(* PLC project Unnamed, Unknown Unnamed 1 *)
(* stored: creationDateTime 2023-06-20T15:59:41, modificationDateTime 2023-06-21T09:28:57 *)

PROGRAM filling_tank
  VAR
    manual AT %QX0.0 : BOOL;
    auto AT %QX0.1 : BOOL;
    emergency_stop AT %QX0.2 : BOOL;
    start AT %QX0.3 : BOOL;
    stop AT %QX0.4 : BOOL;
    reset_button AT %QX0.5 : BOOL;
    start_light AT %QX1.0 : BOOL;
    stop_light AT %QX1.1 : BOOL;
    reset_light AT %QX1.2 : BOOL;
    bottom_valve_open AT %QX1.3 : BOOL;
    top_valve_open AT %QX1.4 : BOOL;
    fictoryioreset AT %QX1.5 : BOOL;
    top_flow AT %QW0 : INT;
    top_level AT %QW1 : INT;
    bottom_flow AT %QW2 : INT;
    bottom_level AT %QW3 : INT;
    top_fill_valve AT %QW4 : INT;
    top_discharge_valve AT %QW5 : INT;
    bottom_fill_valve AT %QW6 : INT;
    bottom_discharge_valve AT %QW7 : INT;
    top_tank AT %QW8 : INT;
    bottom_tank AT %QW9 : INT;
    number_cycles AT %QW10 : INT;
  END_VAR
  VAR
    CTU0 : CTU;
    reset : BOOL;
  END_VAR
  VAR  (* added by the conversion: wires and edge detectors of the diagram *)
    _MOVE9_ENO : BOOL;
    _MOVE9_OUT : INT;
    _LT31_ENO : BOOL;
    _LT31_OUT : BOOL;
    _LT32_ENO : BOOL;
    _LT32_OUT : BOOL;
    _MOVE36_ENO : BOOL;
    _MOVE36_OUT : INT;
    _MOVE38_ENO : BOOL;
    _MOVE38_OUT : INT;
    _GT19_ENO : BOOL;
    _GT19_OUT : BOOL;
    _MOVE22_ENO : BOOL;
    _MOVE22_OUT : INT;
    _MOVE24_ENO : BOOL;
    _MOVE24_OUT : INT;
    _GT49_ENO : BOOL;
    _GT49_OUT : BOOL;
    _MOVE54_ENO : BOOL;
    _MOVE54_OUT : INT;
    _MOVE56_ENO : BOOL;
    _MOVE56_OUT : INT;
    _GT73_ENO : BOOL;
    _GT73_OUT : BOOL;
    _GT81_ENO : BOOL;
    _GT81_OUT : BOOL;
    R_TRIG1 : R_TRIG;
  END_VAR

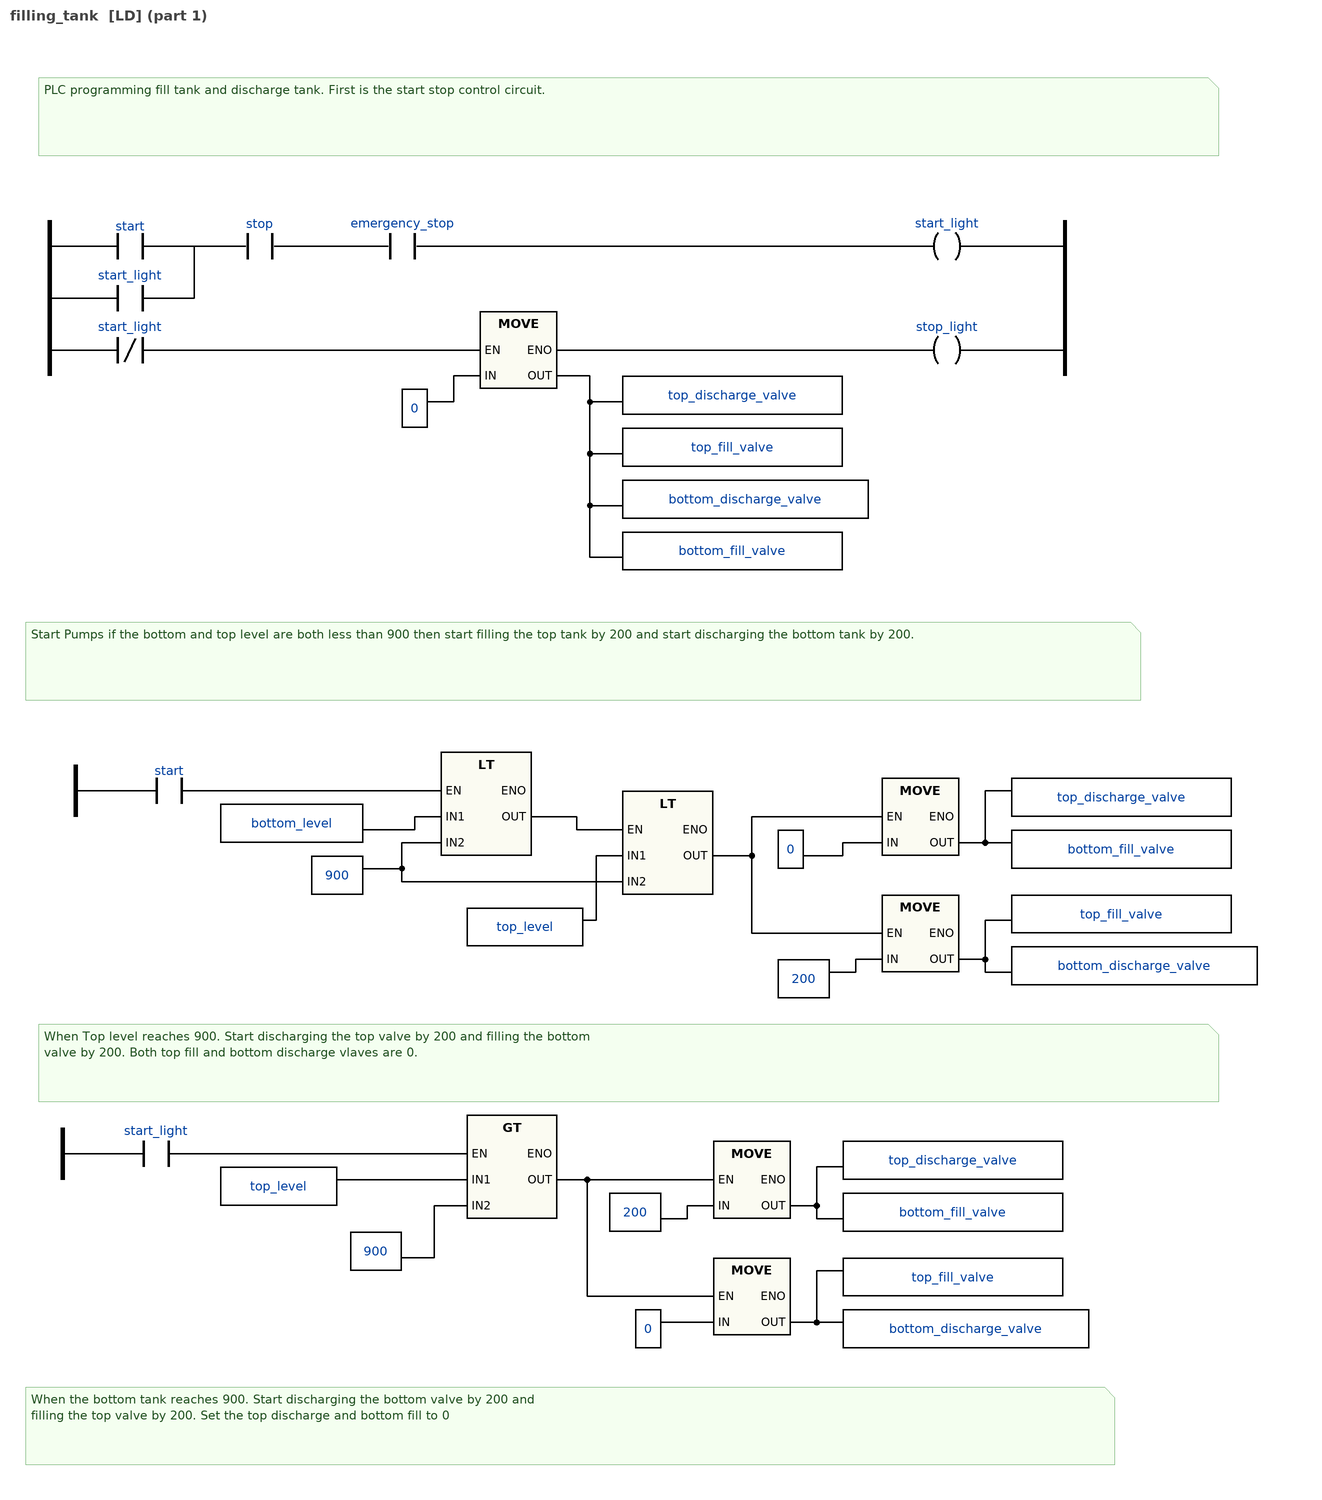
(* LD diagram, written out as Structured Text *)
(* PLC programming fill tank and discharge tank. First is the start stop control circuit. *)
start_light := (start OR start_light) AND stop AND emergency_stop;
_MOVE9_OUT := MOVE(EN := NOT start_light, IN := 0, ENO => _MOVE9_ENO);
stop_light := _MOVE9_ENO;
IF _MOVE9_ENO THEN top_discharge_valve := _MOVE9_OUT; END_IF;
IF _MOVE9_ENO THEN top_fill_valve := _MOVE9_OUT; END_IF;
IF _MOVE9_ENO THEN bottom_discharge_valve := _MOVE9_OUT; END_IF;
IF _MOVE9_ENO THEN bottom_fill_valve := _MOVE9_OUT; END_IF;
(* Start Pumps if the bottom and top level are both less than 900 then start filling the top tank by 200 and start discharging the bottom tank by 200. *)
_LT31_OUT := LT(EN := start, IN1 := bottom_level, IN2 := 900, ENO => _LT31_ENO);
_LT32_OUT := LT(EN := _LT31_OUT, IN1 := top_level, IN2 := 900, ENO => _LT32_ENO);
_MOVE36_OUT := MOVE(EN := _LT32_OUT, IN := 0, ENO => _MOVE36_ENO);
IF _MOVE36_ENO THEN top_discharge_valve := _MOVE36_OUT; END_IF;
IF _MOVE36_ENO THEN bottom_fill_valve := _MOVE36_OUT; END_IF;
_MOVE38_OUT := MOVE(EN := _LT32_OUT, IN := 200, ENO => _MOVE38_ENO);
IF _MOVE38_ENO THEN top_fill_valve := _MOVE38_OUT; END_IF;
IF _MOVE38_ENO THEN bottom_discharge_valve := _MOVE38_OUT; END_IF;
(* When Top level reaches 900. Start discharging the top valve by 200 and filling the bottom 
valve by 200. Both top fill and bottom discharge vlaves are 0. *)
_GT19_OUT := GT(EN := start_light, IN1 := top_level, IN2 := 900, ENO => _GT19_ENO);
_MOVE22_OUT := MOVE(EN := _GT19_OUT, IN := 200, ENO => _MOVE22_ENO);
IF _MOVE22_ENO THEN top_discharge_valve := _MOVE22_OUT; END_IF;
IF _MOVE22_ENO THEN bottom_fill_valve := _MOVE22_OUT; END_IF;
_MOVE24_OUT := MOVE(EN := _GT19_OUT, IN := 0, ENO => _MOVE24_ENO);
IF _MOVE24_ENO THEN top_fill_valve := _MOVE24_OUT; END_IF;
IF _MOVE24_ENO THEN bottom_discharge_valve := _MOVE24_OUT; END_IF;
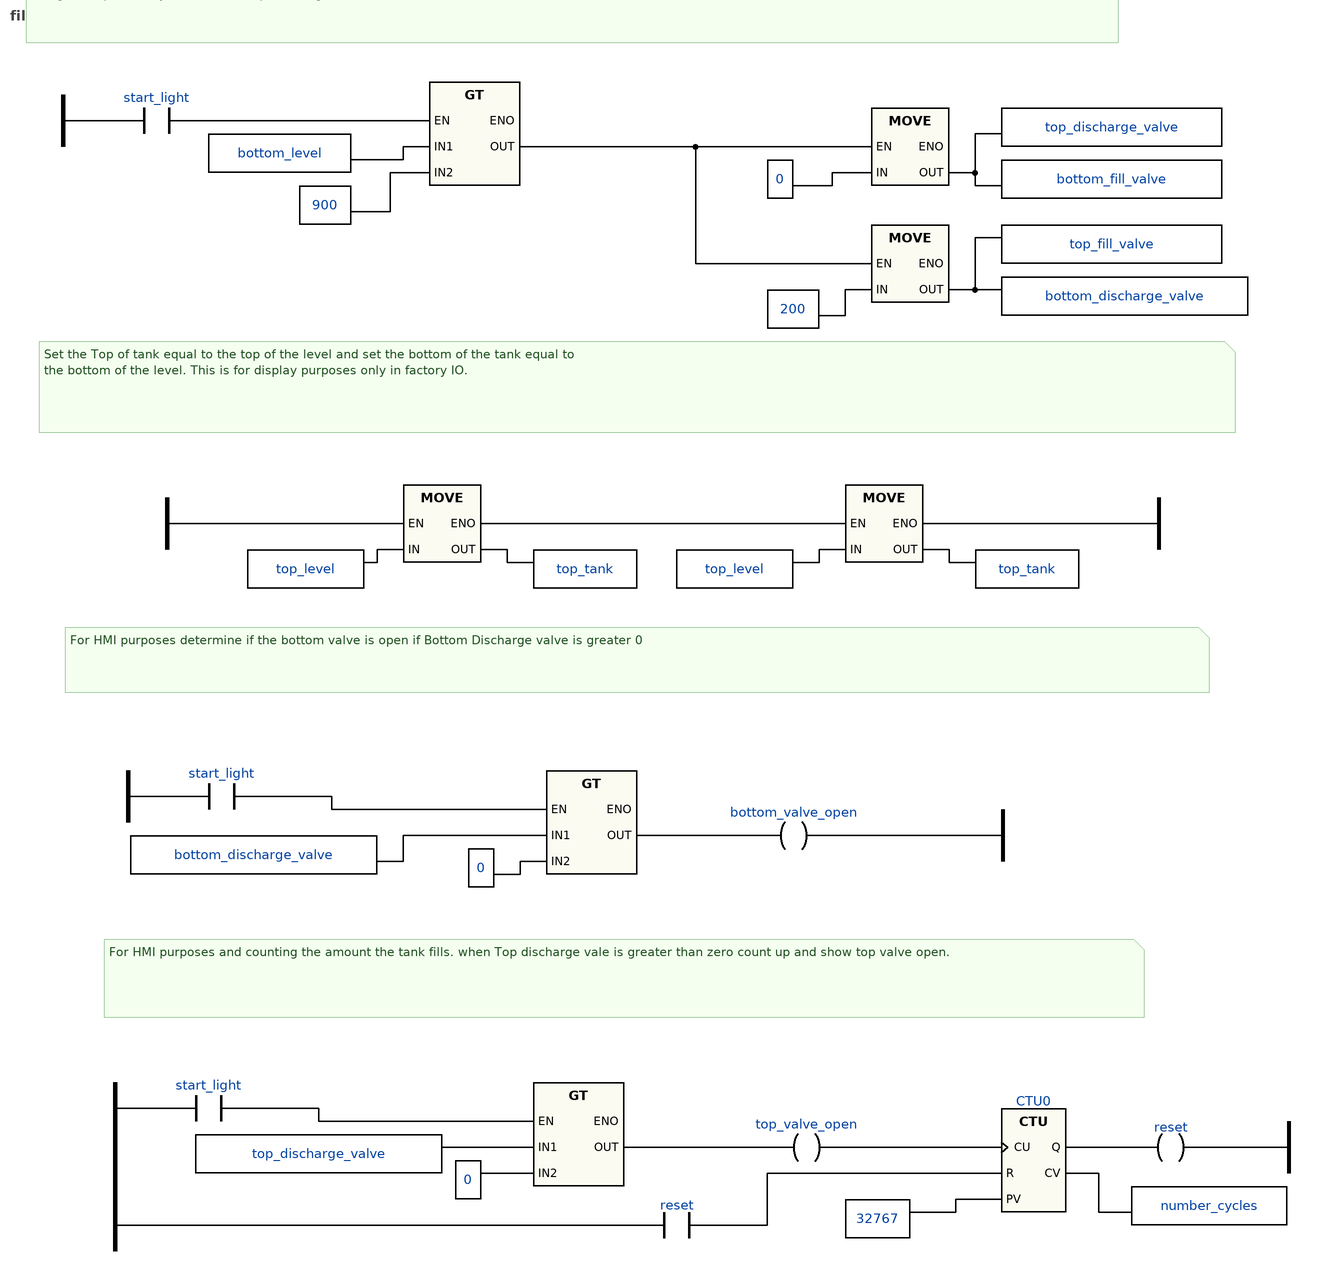
(* When the bottom tank reaches 900. Start discharging the bottom valve by 200 and 
filling the top valve by 200. Set the top discharge and bottom fill to 0 *)
_GT49_OUT := GT(EN := start_light, IN1 := bottom_level, IN2 := 900, ENO => _GT49_ENO);
_MOVE54_OUT := MOVE(EN := _GT49_OUT, IN := 0, ENO => _MOVE54_ENO);
IF _MOVE54_ENO THEN top_discharge_valve := _MOVE54_OUT; END_IF;
IF _MOVE54_ENO THEN bottom_fill_valve := _MOVE54_OUT; END_IF;
_MOVE56_OUT := MOVE(EN := _GT49_OUT, IN := 200, ENO => _MOVE56_ENO);
IF _MOVE56_ENO THEN top_fill_valve := _MOVE56_OUT; END_IF;
IF _MOVE56_ENO THEN bottom_discharge_valve := _MOVE56_OUT; END_IF;
(* Set the Top of tank equal to the top of the level and set the bottom of the tank equal to
 the bottom of the level. This is for display purposes only in factory IO. *)
top_tank := top_level;
top_tank := top_level;
(* For HMI purposes determine if the bottom valve is open if Bottom Discharge valve is greater 0 *)
_GT73_OUT := GT(EN := start_light, IN1 := bottom_discharge_valve, IN2 := 0, ENO => _GT73_ENO);
bottom_valve_open := _GT73_OUT;
(* For HMI purposes and counting the amount the tank fills. when Top discharge vale is greater than zero count up and show top valve open. *)
_GT81_OUT := GT(EN := start_light, IN1 := top_discharge_valve, IN2 := 0, ENO => _GT81_ENO);
top_valve_open := _GT81_OUT;
R_TRIG1(CLK := _GT81_OUT);
CTU0(CU := R_TRIG1.Q, R := reset, PV := 32767);
reset := CTU0.Q;
number_cycles := CTU0.CV;
END_PROGRAM

CONFIGURATION Config0
  RESOURCE Res0 ON PLC
    TASK task0(INTERVAL := T#20ms, PRIORITY := 0);
    PROGRAM instance0 WITH task0 : filling_tank;
  END_RESOURCE
END_CONFIGURATION
